# EPICS autosave request: PEARLCAM/iocBoot/iocPEARLCAM-IOC-01/WEBCAM_01_settings.req
file "URLDriver_settings.req",      P=$(P),  R=CAM1:
#file "NDStdArrays_settings.req",    P=$(P),  R=ROI1:
